// TIA Portal V20 export
// export: Created 2025-12-01T14:57:43.5258514Z, ExportSetting None, DisplayName Totally Integrated Automation Portal, DisplayVersion V20 Update 3, DisplayName TIA Portal Openness, DisplayVersion V20 Update 3, DisplayName TIA Portal Version Control Interface, DisplayVersion V20 Update 3, DisplayName STEP 7 Professional, DisplayVersion V20 Update 3, DisplayName STEP 7 Safety, DisplayVersion V20 Update 2, DisplayName WinCC Basic/Comfort/Advanced, DisplayVersion V20 Update 3, DisplayName WinCC Professional, DisplayVersion V20 Update 3, DisplayName WinCC Unified, DisplayVersion V20 Update 3
FUNCTION "FC504_SIM_Ordenes_Desvios_SCR" : Void   // FC504, LAD
{ S7_Optimized_Access := 'FALSE' }
AUTHOR : ROUTER
NAME : 20190911
VERSION : 3.1
// stored: AutoNumber false, SetENOAutomatically false
   VAR_INPUT
      Sacar_orden : Bool;
      Reset : Bool;
      Bandejas_S3 : UDInt;
      Bandejas_S2 : UDInt;
   END_VAR
   VAR_OUTPUT
      Orden_FIFO : "ROUT_Orden_Fifo_Scanner";
   END_VAR
   VAR_IN_OUT
      Mem_FP : Bool;
      Aux_CNT : UDInt;
   END_VAR
   VAR_TEMP
      relleno : Byte;
      retval : Int;
      Suma_Bandejas_totales : UDInt;
      Bandejas_S3_menos1 : UDInt;
   END_VAR
   VAR_TEMP   // added for the SCL form of the ladder/FBD networks
      _w1 : Bool;
      _w2 : Bool;
   END_VAR
BEGIN

REGION Network 1
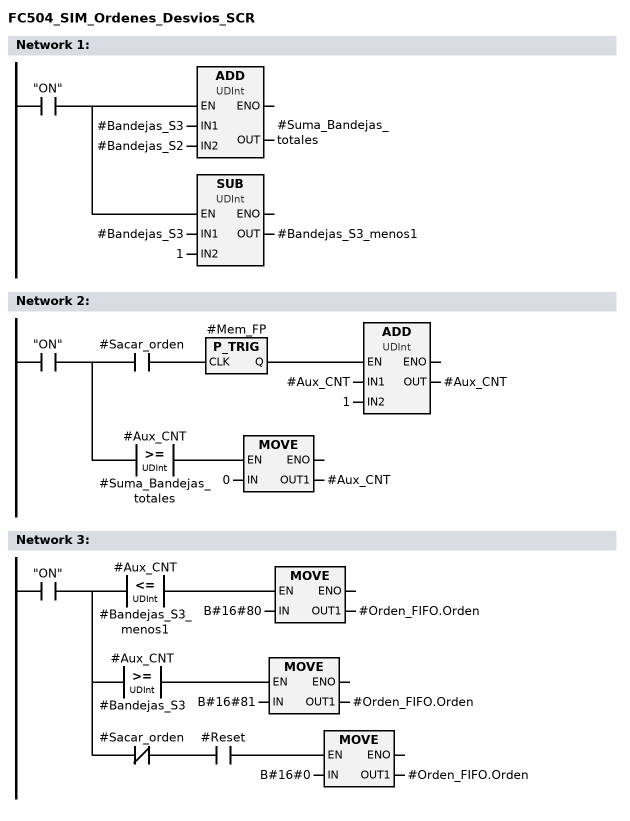
   RUNG wire#powerrail
      Contact( "ON" )
      wire#w1
      { S7_Templates := "SrcType := UDInt"; S7_GenerateENO := "TRUE" } Add(in1 := #Bandejas_S3, in2 := #Bandejas_S2, out => #Suma_Bandejas_totales)
   END_RUNG
   RUNG wire#w1
      { S7_Templates := "SrcType := UDInt"; S7_GenerateENO := "TRUE" } Sub(in1 := #Bandejas_S3, in2 := 1, out => #Bandejas_S3_menos1)
   END_RUNG
   // the same network as SCL:
   IF "ON" THEN
       #Suma_Bandejas_totales := #Bandejas_S3 + #Bandejas_S2;
       #Bandejas_S3_menos1 := #Bandejas_S3 - 1;
   END_IF;
END_REGION

REGION Network 2
   RUNG wire#powerrail
      Contact( "ON" )
      wire#w1
      Contact( #Sacar_orden )
      P_Trig( #Mem_FP )
      { S7_Templates := "SrcType := UDInt"; S7_GenerateENO := "TRUE" } Add(in1 := #Aux_CNT, in2 := 1, out => #Aux_CNT)
   END_RUNG
   RUNG wire#w1
      { S7_Templates := "SrcType := UDInt" } GE_Contact(in1 := #Aux_CNT, in2 := #Suma_Bandejas_totales)
      { S7_GenerateENO := "TRUE" } Move(in := 0, out1 => #Aux_CNT)
   END_RUNG
   // the same network as SCL:
   #_w1 := "ON" AND #Sacar_orden;
   #_w2 := #_w1 AND NOT #Mem_FP;   // rising edge
   #Mem_FP := #_w1;
   IF #_w2 THEN #Aux_CNT := #Aux_CNT + 1; END_IF;
   IF "ON" AND (#Aux_CNT >= #Suma_Bandejas_totales) THEN #Aux_CNT := 0; END_IF;
END_REGION

REGION Network 3
   RUNG wire#powerrail
      Contact( "ON" )
      wire#w1
      { S7_Templates := "SrcType := UDInt" } LE_Contact(in1 := #Aux_CNT, in2 := #Bandejas_S3_menos1)
      { S7_GenerateENO := "TRUE" } Move(in := B#16#80, out1 => #Orden_FIFO.Orden)
   END_RUNG
   RUNG wire#w1
      { S7_Templates := "SrcType := UDInt" } GE_Contact(in1 := #Aux_CNT, in2 := #Bandejas_S3)
      { S7_GenerateENO := "TRUE" } Move(in := B#16#81, out1 => #Orden_FIFO.Orden)
   END_RUNG
   RUNG wire#w1
      I_Contact( #Sacar_orden )
      Contact( #Reset )
      { S7_GenerateENO := "TRUE" } Move(in := B#16#0, out1 => #Orden_FIFO.Orden)
   END_RUNG
   // the same network as SCL:
   IF "ON" AND (#Aux_CNT <= #Bandejas_S3_menos1) THEN #Orden_FIFO.Orden := B#16#80; END_IF;
   IF "ON" AND (#Aux_CNT >= #Bandejas_S3) THEN #Orden_FIFO.Orden := B#16#81; END_IF;
   IF "ON" AND NOT #Sacar_orden AND #Reset THEN #Orden_FIFO.Orden := B#16#0; END_IF;
END_REGION
END_FUNCTION
